// TwinCAT 3 PLC project test
// ProgramVersion: 3.1.4020.5
// libraries:
//   LCLS General, * (SLAC)
//   LCLS Vacuum, * (SLAC - LCLS)
//   PMPS, * (SLAC - LCLS)
//   Tc2_Standard, * (Beckhoff Automation GmbH)
//   Tc2_System, * (Beckhoff Automation GmbH)
//   Tc2_Utilities, * (Beckhoff Automation GmbH)
//   Tc3_Module, * (Beckhoff Automation GmbH)
// project tree:
//   DUTs/ E_STATES.TcTLEO (not stored)
//   functions/ FB_TurboExtLogic.TcPOU, F_RoughPumpInlet_ILK.TcPOU, F_TurboExtILKLogic.TcPOU, F_TurboExtILKLogic_2.TcPOU, F_TurboExtILK_NO.TcPOU, F_TurboExtILK_NO_T.TcPOU, F_TurboGateValve_ILK.TcPOU, F_TurboGateValve_ILK_1.TcPOU (not stored), F_TurboGateValve_Protection_ILK.TcPOU, F_TURBO_VRC_ILK.TcPOU, F_VALVE_REL_ILK.TcPOU (not stored), F_VRC_DIODE_ILK.TcPOU, F_VRC_DIODE_ILK_OK.TcPOU
//   GVLs/ GVL_Devices.TcGVL, GVL_PMPS.TcGVL
//   / PlcTask.TcTTO (not stored)
//   POUs/ FB_VGC_tst.TcPOU, MAIN.TcPOU
// real-time tasks:
//   TASK PlcTask: cycle T#10ms, priority 20, ADS port 350
//   TASK SimTask: cycle T#10ms, priority 1, ADS port 351
//   TASK VacTask: cycle T#10ms, priority 2, ADS port 352
// I/O:
//   DEVICE Device 1 (EtherCAT) (disabled), AmsNetId 172.21.148.60.2.1
//     Term 1 (EK1100) [EK1100 EtherCAT Coupler (2A E-Bus)]
//       Term 2 (EL3174-0002) [EL3174-0002 4Ch. Ana. Input +/-10V, +/-20mA 16 Bit, Isolated Channels]
//       Term 3 (EL3174-0002) [EL3174-0002 4Ch. Ana. Input +/-10V, +/-20mA 16 Bit, Isolated Channels]
//       Term 4 (EL2624) [EL2624 4Ch. Relay Output, NO (125V AC / 30V DC)]
//       Term 6 (EL1004) [EL1004 4Ch. Dig. Input 24V, 3ms]
//       Term 5 (EL1004) [EL1004 4Ch. Dig. Input 24V, 3ms]
//       Term 7 (EL2004) [EL2004 4Ch. Dig. Output 24V, 0.5A]
//       Term 8 (EL3064) [EL3064 4Ch. Ana. Input 0-10V]
//       Term 9 (EL2794) [EL2794 4Ch. Dig. Output 24V AC/DC, 2A, short-circuit-proof]
//       Term 10 (EL1004) [EL1004 4Ch. Dig. Input 24V, 3ms]
//       Term 11 (EL1124) [EL1124 4Ch. Dig. Input 5V, 10µs, Sensor Power]
//       Term 12 (EL1124) [EL1124 4Ch. Dig. Input 5V, 10µs, Sensor Power]
//       Term 13 (EL3064) [EL3064 4Ch. Ana. Input 0-10V]
// variable links:
//   SIM/SIM Instance <-> test/test Instance
//     PlcTaskSim Inputs/GVL_SimDevices.PMPS_VGC_01.i_xSol <-> PlcTask Outputs/GVL_Devices.PMPS_VGC_01.q_xOPN_DO
//     PlcTaskSim Inputs/GVL_SimDevices.PMPS_VGC_02.i_xSol <-> PlcTask Outputs/GVL_Devices.PMPS_VGC_02.q_xOPN_DO
//     PlcTaskSim Inputs/GVL_SimDevices.PMPS_VGC_03.i_xSol <-> PlcTask Outputs/GVL_Devices.PMPS_VGC_03.q_xOPN_DO
//     PlcTaskSim Inputs/GVL_SimDevices.PMPS_VGC_04.i_xSol <-> PlcTask Outputs/GVL_Devices.PMPS_VGC_04.q_xOPN_DO
//     PlcTaskSim Inputs/GVL_SimDevices.PMPS_VGC_05.i_xSol <-> PlcTask Outputs/GVL_Devices.PMPS_VGC_05.q_xOPN_DO
//     PlcTaskSim Inputs/GVL_SimDevices.PMPS_VGC_06.i_xSol <-> PlcTask Outputs/GVL_Devices.PMPS_VGC_06.q_xOPN_DO
//     PlcTaskSim Inputs/GVL_SimDevices.PMPS_VGC_08.i_xSol <-> PlcTask Outputs/GVL_Devices.PMPS_VGC_08.q_xOPN_DO
//     PlcTaskSim Inputs/GVL_SimDevices.PMPS_VGC_09.i_xSol <-> PlcTask Outputs/GVL_Devices.PMPS_VGC_09.q_xOPN_DO
//     PlcTaskSim Inputs/GVL_SimDevices.PMPS_VGC_10.i_xSol <-> PlcTask Outputs/GVL_Devices.PMPS_VGC_10.q_xOPN_DO
//     PlcTaskSim Inputs/GVL_SimDevices.PMPS_VGC_11.i_xSol <-> PlcTask Outputs/GVL_Devices.PMPS_VGC_11.q_xOPN_DO
//     PlcTaskSim Inputs/GVL_SimDevices.S_FEE_GCC_03.i_xHvOn <-> PlcTask Outputs/GVL_Devices.FEE_GCC_03.q_xHV_DIS
//     PlcTaskSim Inputs/GVL_SimDevices.S_FEE_GCC_04.i_xHvOn <-> PlcTask Outputs/GVL_Devices.FEE_GCC_04.q_xHV_DIS
//     PlcTaskSim Inputs/GVL_SimDevices.S_FEE_KMONO_GCC_01.i_xHvOn <-> PlcTask Outputs/GVL_Devices.FEE_KMONO_GCC_01.q_xHV_DIS
//     PlcTaskSim Inputs/GVL_SimDevices.S_FEE_KMONO_PIP_01.xOn <-> PlcTask Outputs/GVL_Devices.FEE_KMONO_PIP_01.q_xHVEna_DO
//     PlcTaskSim Inputs/GVL_SimDevices.S_FEE_M1L_PIP_01.xOn <-> PlcTask Outputs/GVL_Devices.FEE_M1L_PIP_01.q_xHVEna_DO
//     PlcTaskSim Inputs/GVL_SimDevices.S_FEE_MIL_GCC_02.i_xHvOn <-> PlcTask Outputs/GVL_Devices.FEE_M1L_GCC_01.q_xHV_DIS
//     PlcTaskSim Inputs/GVL_SimDevices.S_FEE_PIP_02.xOn <-> PlcTask Outputs/GVL_Devices.FEE_PIP_02.q_xHVEna_DO
//     PlcTaskSim Inputs/GVL_SimDevices.S_FEE_PIP_03.xOn <-> PlcTask Outputs/GVL_Devices.FEE_PIP_03.q_xHVEna_DO
//     PlcTaskSim Inputs/GVL_SimDevices.S_FEE_VGC_02.i_xSol <-> PlcTask Outputs/GVL_Devices.FEE_VGC_02.q_xOPN_DO
//     PlcTaskSim Inputs/GVL_SimDevices.VGC_2S.i_xSol <-> PlcTask Outputs/MAIN.VGC_2S.q_xOPN_DO
//     PlcTaskSim Outputs/GVL_SimDevices.PMPS_VGC_01.q_xClsLS <-> PlcTask Inputs/GVL_Devices.PMPS_VGC_01.i_xClsLS
//     PlcTaskSim Outputs/GVL_SimDevices.PMPS_VGC_02.q_xClsLS <-> PlcTask Inputs/GVL_Devices.PMPS_VGC_02.i_xClsLS
//     PlcTaskSim Outputs/GVL_SimDevices.PMPS_VGC_03.q_xClsLS <-> PlcTask Inputs/GVL_Devices.PMPS_VGC_03.i_xClsLS
//     PlcTaskSim Outputs/GVL_SimDevices.PMPS_VGC_04.q_xClsLS <-> PlcTask Inputs/GVL_Devices.PMPS_VGC_04.i_xClsLS
//     PlcTaskSim Outputs/GVL_SimDevices.PMPS_VGC_05.q_xClsLS <-> PlcTask Inputs/GVL_Devices.PMPS_VGC_05.i_xClsLS
//     PlcTaskSim Outputs/GVL_SimDevices.PMPS_VGC_06.q_xClsLS <-> PlcTask Inputs/GVL_Devices.PMPS_VGC_06.i_xClsLS
//     PlcTaskSim Outputs/GVL_SimDevices.PMPS_VGC_08.q_xClsLS <-> PlcTask Inputs/GVL_Devices.PMPS_VGC_08.i_xClsLS
//     PlcTaskSim Outputs/GVL_SimDevices.PMPS_VGC_09.q_xClsLS <-> PlcTask Inputs/GVL_Devices.PMPS_VGC_09.i_xClsLS
//     PlcTaskSim Outputs/GVL_SimDevices.PMPS_VGC_10.q_xClsLS <-> PlcTask Inputs/GVL_Devices.PMPS_VGC_10.i_xClsLS
//     PlcTaskSim Outputs/GVL_SimDevices.PMPS_VGC_11.q_xClsLS <-> PlcTask Inputs/GVL_Devices.PMPS_VGC_11.i_xClsLS
//     PlcTaskSim Outputs/GVL_SimDevices.PMPS_VGC_01.q_xOpnLS <-> PlcTask Inputs/GVL_Devices.PMPS_VGC_01.i_xOpnLS
//     PlcTaskSim Outputs/GVL_SimDevices.PMPS_VGC_02.q_xOpnLS <-> PlcTask Inputs/GVL_Devices.PMPS_VGC_02.i_xOpnLS
//     PlcTaskSim Outputs/GVL_SimDevices.PMPS_VGC_03.q_xOpnLS <-> PlcTask Inputs/GVL_Devices.PMPS_VGC_03.i_xOpnLS
//     PlcTaskSim Outputs/GVL_SimDevices.PMPS_VGC_04.q_xOpnLS <-> PlcTask Inputs/GVL_Devices.PMPS_VGC_04.i_xOpnLS
//     PlcTaskSim Outputs/GVL_SimDevices.PMPS_VGC_05.q_xOpnLS <-> PlcTask Inputs/GVL_Devices.PMPS_VGC_05.i_xOpnLS
//     PlcTaskSim Outputs/GVL_SimDevices.PMPS_VGC_06.q_xOpnLS <-> PlcTask Inputs/GVL_Devices.PMPS_VGC_06.i_xOpnLS
//     PlcTaskSim Outputs/GVL_SimDevices.PMPS_VGC_08.q_xOpnLS <-> PlcTask Inputs/GVL_Devices.PMPS_VGC_08.i_xOpnLS
//     PlcTaskSim Outputs/GVL_SimDevices.PMPS_VGC_09.q_xOpnLS <-> PlcTask Inputs/GVL_Devices.PMPS_VGC_09.i_xOpnLS
//     PlcTaskSim Outputs/GVL_SimDevices.PMPS_VGC_10.q_xOpnLS <-> PlcTask Inputs/GVL_Devices.PMPS_VGC_10.i_xOpnLS
//     PlcTaskSim Outputs/GVL_SimDevices.PMPS_VGC_11.q_xOpnLS <-> PlcTask Inputs/GVL_Devices.PMPS_VGC_11.i_xOpnLS
//     PlcTaskSim Outputs/GVL_SimDevices.S_FEE_GCC_03.q_DisActive <-> PlcTask Inputs/GVL_Devices.FEE_GCC_03.i_xDisc_Active
//     PlcTaskSim Outputs/GVL_SimDevices.S_FEE_GCC_04.q_DisActive <-> PlcTask Inputs/GVL_Devices.FEE_GCC_04.i_xDisc_Active
//     PlcTaskSim Outputs/GVL_SimDevices.S_FEE_GCC_03.q_iRawPress <-> PlcTask Inputs/GVL_Devices.FEE_GCC_03.i_iPRESS_R
//     PlcTaskSim Outputs/GVL_SimDevices.S_FEE_GCC_04.q_iRawPress <-> PlcTask Inputs/GVL_Devices.FEE_GCC_04.i_iPRESS_R
//     PlcTaskSim Outputs/GVL_SimDevices.S_FEE_GCC_03.q_xHVOn <-> PlcTask Inputs/GVL_Devices.FEE_GCC_03.i_xHV_ON
//     PlcTaskSim Outputs/GVL_SimDevices.S_FEE_GCC_04.q_xHVOn <-> PlcTask Inputs/GVL_Devices.FEE_GCC_04.i_xHV_ON
//     PlcTaskSim Outputs/GVL_SimDevices.S_FEE_GPI_03.q_iRawPress <-> PlcTask Inputs/GVL_Devices.FEE_GPI_03.i_iPRESS_R
//     PlcTaskSim Outputs/GVL_SimDevices.S_FEE_GPI_04.q_iRawPress <-> PlcTask Inputs/GVL_Devices.FEE_GPI_04.i_iPRESS_R
//     PlcTaskSim Outputs/GVL_SimDevices.S_FEE_KMONO_GCC_01.q_DisActive <-> PlcTask Inputs/GVL_Devices.FEE_KMONO_GCC_01.i_xDisc_Active
//     PlcTaskSim Outputs/GVL_SimDevices.S_FEE_KMONO_GCC_01.q_iRawPress <-> PlcTask Inputs/GVL_Devices.FEE_KMONO_GCC_01.i_iPRESS_R
//     PlcTaskSim Outputs/GVL_SimDevices.S_FEE_KMONO_GCC_01.q_xHVOn <-> PlcTask Inputs/GVL_Devices.FEE_KMONO_GCC_01.i_xHV_ON
//     PlcTaskSim Outputs/GVL_SimDevices.S_FEE_KMONO_GPI_01.q_iRawPress <-> PlcTask Inputs/GVL_Devices.FEE_KMONO_GPI_01.i_iPRESS_R
//     PlcTaskSim Outputs/GVL_SimDevices.S_FEE_M1L_GPI_02.q_iRawPress <-> PlcTask Inputs/GVL_Devices.FEE_M1L_GPI_01.i_iPRESS_R
//     PlcTaskSim Outputs/GVL_SimDevices.S_FEE_MIL_GCC_02.q_DisActive <-> PlcTask Inputs/GVL_Devices.FEE_M1L_GCC_01.i_xDisc_Active
//     PlcTaskSim Outputs/GVL_SimDevices.S_FEE_MIL_GCC_02.q_iRawPress <-> PlcTask Inputs/GVL_Devices.FEE_M1L_GCC_01.i_iPRESS_R
//     PlcTaskSim Outputs/GVL_SimDevices.S_FEE_MIL_GCC_02.q_xHVOn <-> PlcTask Inputs/GVL_Devices.FEE_M1L_GCC_01.i_xHV_ON
//     PlcTaskSim Outputs/GVL_SimDevices.S_FEE_VGC_02.q_xClsLS <-> PlcTask Inputs/GVL_Devices.FEE_VGC_02.i_xClsLS
//     PlcTaskSim Outputs/GVL_SimDevices.S_FEE_VGC_02.q_xOpnLS <-> PlcTask Inputs/GVL_Devices.FEE_VGC_02.i_xOpnLS
//     PlcTaskSim Outputs/GVL_SimDevices.VGC_2S.q_xClsLS <-> PlcTask Inputs/MAIN.VGC_2S.i_xClsLS
//     PlcTaskSim Outputs/GVL_SimDevices.VGC_2S.q_xOpnLS <-> PlcTask Inputs/MAIN.VGC_2S.i_xOpnLS

// ---- GVLs/GVL_Devices.TcGVL
VAR_GLOBAL
	
	

/////////////////////
	{attribute 'pytmc' := '
    pv: FEE:VGC:02
	'}
	FEE_VGC_02: FB_VGC;
	{attribute 'pytmc' := '
    pv: FEE:KMONO:GPI:01
	'}
	FEE_KMONO_GPI_01: FB_MKS275;
	{attribute 'pytmc' := '
    pv: FEE:KMONO:GCC:01
	'}
	FEE_KMONO_GCC_01: FB_MKS500;
	{attribute 'pytmc' := '
    pv: FEE:KMONO:PIP:01
	'}
	FEE_KMONO_PIP_01: FB_PIP_Gamma;
	{attribute 'pytmc' := '
    pv: FEE:PIP:02
	'}
	FEE_PIP_02: FB_PIP_Gamma;
	{attribute 'pytmc' := '
    pv: FEE:GPI:03
	'}
	FEE_GPI_03: FB_MKS275;
	{attribute 'pytmc' := '
    pv: FEE:GCC:03
	'}
	FEE_GCC_03: FB_MKS500;
	{attribute 'pytmc' := '
    pv: FEE:VGC:03
	'}
	//FEE_VGC_03: FB_VGC_FFO;
	{attribute 'pytmc' := '
    pv: FEE:M1L:GPI:01
	'}
	FEE_M1L_GPI_01: FB_MKS275;
	{attribute 'pytmc' := '
    pv: FEE:M1L:GCC:03
	'}
	FEE_M1L_GCC_01: FB_MKS500;
	{attribute 'pytmc' := '
    pv: FEE:M1L:PIP:01
	'}
	FEE_M1L_PIP_01: FB_PIP_Gamma;
	{attribute 'pytmc' := '
    pv: FEE:PIP:03
	'}
	FEE_PIP_03: FB_PIP_Gamma;
	{attribute 'pytmc' := '
    pv: FEE:GPI:04
	'}
	FEE_GPI_04: FB_MKS275;
	{attribute 'pytmc' := '
    pv: FEE:GCC:04
	'}
	FEE_GCC_04: FB_MKS500;
	{attribute 'pytmc' := '
    pv: FEE:VGC:04
	'}
	//FEE_VGC_04: FB_VGC_FFO;
	
	PMPS_VGC_01: FB_VGC;
	PMPS_VGC_02: FB_VGC;
	PMPS_VGC_03: FB_VGC;
	PMPS_VGC_04: FB_VGC;
	PMPS_VGC_05: FB_VGC;
	PMPS_VGC_06: FB_VGC;
	
	PMPS_VGC_08: FB_VGC;
	PMPS_VGC_09: FB_VGC;
	
	PMPS_VGC_10: FB_VGC;
	PMPS_VGC_11: FB_VGC;
	
	PTM_Agilent: FB_PTM_Agilent; 
			
	
END_VAR

// ---- GVLs/GVL_PMPS.TcGVL

VAR_GLOBAL
	 g_FastFaultOutput3  :   FB_HardwareFFOutput;
	
{attribute 'pytmc' := '
    pv: PLC:TST:FF1
    '}
    {attribute 'TcLinkTo' := '.q_xFastFaultOut:=TIIB[PMPS_FFO]^Channel 1^Output'}
    g_FastFaultOutput1  :   FB_HardwareFFOutput;
	
	{attribute 'pytmc' := '
    pv: PLC:TST:FF2
    '}
    {attribute 'TcLinkTo' := '.q_xFastFaultOut:=TIIB[PMPS_FFO]^Channel 2^Output'}
    g_FastFaultOutput2  :   FB_HardwareFFOutput;
	
END_VAR

// ---- functions/FB_TurboExtLogic.TcPOU
(*deprecated*)
FUNCTION_BLOCK FB_TurboExtLogic
VAR_IN_OUT
	Turbo		:	ST_AgilentPTM;
END_VAR
VAR_INPUT
	BackingGauge:	ST_VG;
	InletGauge	:	ST_VG;
	VentValve	:	ST_VCC_NO;
	ScrollPump	:	ST_RoughPump;
END_VAR
VAR_OUTPUT
END_VAR
VAR
END_VAR

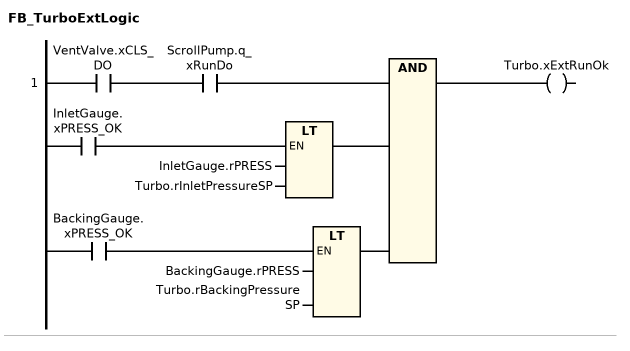
// NETWORK 1
Turbo.xExtRunOk := (VentValve.xCLS_DO AND ScrollPump.q_xRunDo) AND (InletGauge.xPRESS_OK AND InletGauge.rPRESS < Turbo.rInletPressureSP) AND (BackingGauge.xPRESS_OK AND BackingGauge.rPRESS < Turbo.rBackingPressureSP);

END_FUNCTION_BLOCK

// ---- functions/F_RoughPumpInlet_ILK.TcPOU
(*
	Determine whether a pump attached to the inlet of a roughing pump is safe to open. 
	
	Return true, signaling it is safe to open when the roughing pump is confirmed to be working. 
*)

FUNCTION F_RoughPumpInlet_ILK : BOOL
VAR_INPUT
	ScrollPump	:	ST_RoughPump;
END_VAR
VAR
END_VAR


F_RoughPumpInlet_ILK := (ScrollPump.eState = pumpRUNNING); (* Confirm that the roughing pump is running before opening the valve *)

END_FUNCTION

// ---- functions/F_TurboExtILKLogic.TcPOU

(* This function evaluates the Turbo ILK logic*)
(* The Turbo shall not Run if the vent valve is open*)
(* The function also switches off the Turbo if the Inlet pressure or the backing Pressure*)
(* are higher than the configured set point*)
FUNCTION F_TurboExtILKLogic : BOOL
VAR_INPUT
	Turbo		:	ST_PTM;
	BackingGauge:	ST_VG;
	InletGauge	:	ST_VG;
	VentValve	:	ST_VVC;
	ScrollPump	:	ST_RoughPump;
END_VAR

VAR
END_VAR

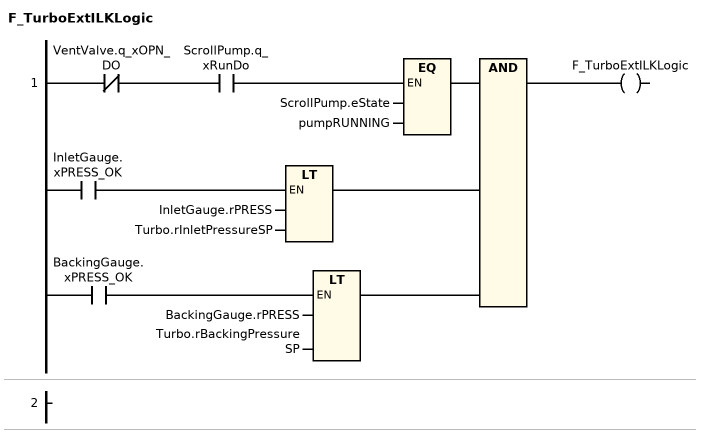
// NETWORK 1
F_TurboExtILKLogic := (NOT VentValve.q_xOPN_DO AND ScrollPump.q_xRunDo AND ScrollPump.eState = pumpRUNNING) AND (InletGauge.xPRESS_OK AND InletGauge.rPRESS < Turbo.rInletPressureSP) AND (BackingGauge.xPRESS_OK AND BackingGauge.rPRESS < Turbo.rBackingPressureSP);

// NETWORK 2

END_FUNCTION

// ---- functions/F_TurboExtILKLogic_2.TcPOU

(* This function evaluates the Turbo ILK logic*)
(* The function switches off the Turbo if the Inlet pressure or the backing Pressure*)
(* are higher than the configured set point*)
FUNCTION F_TurboExtILKLogic_2 : BOOL
VAR_INPUT
	Turbo		:	ST_PTM;
	BackingGauge:	ST_VG;
	InletGauge	:	ST_VG;
	ScrollPump	:	ST_RoughPump;
END_VAR
VAR
END_VAR

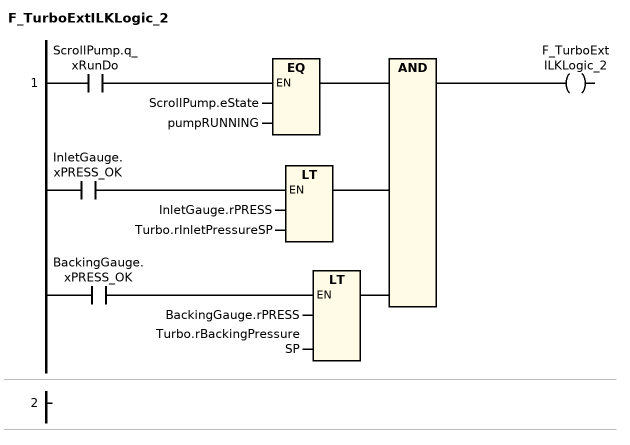
// NETWORK 1
F_TurboExtILKLogic_2 := (ScrollPump.q_xRunDo AND ScrollPump.eState = pumpRUNNING) AND (InletGauge.xPRESS_OK AND InletGauge.rPRESS < Turbo.rInletPressureSP) AND (BackingGauge.xPRESS_OK AND BackingGauge.rPRESS < Turbo.rBackingPressureSP);

// NETWORK 2

END_FUNCTION

// ---- functions/F_TurboExtILK_NO.TcPOU
(* This function Block interfaces with a NO turbo valve*)
(* Mainly used in the FEE HXR GATT*)
FUNCTION F_TurboExtILK_NO : BOOL
VAR_INPUT
	Turbo		:	ST_PTM;
	BackingGauge:	ST_VG;
	InletGauge	:	ST_VG;
	VentValve	:	ST_VCC_NO; //NO type turbo valve
	ScrollPump	:	ST_RoughPump;
	Timer :TON;
END_VAR

VAR
END_VAR
VAR // added by the converter: edge detectors and wires of the graphical bodies
    _w1 : BOOL;
END_VAR

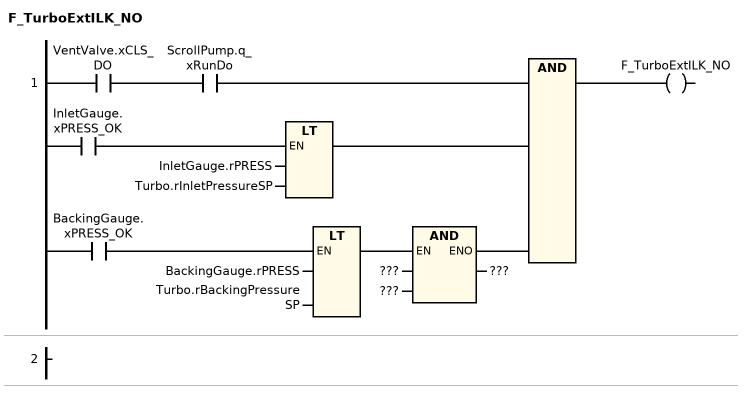
// NETWORK 1
_w1 := BackingGauge.xPRESS_OK AND BackingGauge.rPRESS < Turbo.rBackingPressureSP;
IF _w1 THEN (* ??? AND ???; result not used *) END_IF
F_TurboExtILK_NO := (VentValve.xCLS_DO AND ScrollPump.q_xRunDo) AND (InletGauge.xPRESS_OK AND InletGauge.rPRESS < Turbo.rInletPressureSP) AND _w1;

// NETWORK 2

END_FUNCTION

// ---- functions/F_TurboExtILK_NO_T.TcPOU
FUNCTION F_TurboExtILK_NO_T : BOOL
VAR_INPUT
	Turbo		:	ST_PTM;
	BackingGauge:	ST_VG;
	InletGauge	:	ST_VG;
	VentValve	:	ST_VCC_NO; //NO type turbo valve
	ScrollPump	:	ST_RoughPump;
END_VAR
VAR
	Timer :TON;
END_VAR

END_FUNCTION

// ---- functions/F_TurboGateValve_ILK.TcPOU
(* This Function Block evaluates the ILK condition of the Turbo Gate valve *)
(* The logic Protects the Turbo pump from inlet pressure above the SP*)

FUNCTION F_TurboGateValve_ILK : BOOL (* function return TRUE when ILK is OK*)
VAR_INPUT
	i_Turbo : ST_PTM; // Turbo Pump
	i_stISG : ST_VG; //Gauge measuring inlet Pressure e.g Pirani
END_VAR
VAR
END_VAR

(* This Function Block evaluates the ILK condition of the Turbo Gate valve *)
(* The logic Protects the Turbo pump from inlet pressure above the SP*)
F_TurboGateValve_ILK := (NOT (i_Turbo.eState = pumpSTOPPED) AND NOT (i_Turbo.eState = pumpSTOPPING) AND NOT (i_Turbo.eState = pumpFAULT))
						AND (i_stISG.xPRESS_OK AND i_stISG.rPRESS < i_Turbo.rInletPressureSP);

END_FUNCTION

// ---- functions/F_TurboGateValve_Protection_ILK.TcPOU
(* This Function Block evaluates the ILK condition of the Turbo Gate valve *)
(* The logic Protects the Turbo pump from inlet pressure above the SP*)
(* And Protects the Turbo pump from backing pressure above the SP*)
(* And Protects the Turbo pump in the case of backing pump not running*)

FUNCTION F_TurboGateValve_Protection_ILK : BOOL (* function return TRUE when ILK is OK*)
VAR_INPUT
	i_Turbo : ST_PTM; // Turbo Pump
	i_stISG : ST_VG; //Gauge measuring inlet Pressure e.g Pirani
	i_stBSG : ST_VG; //Gauge measuring backing Pressure e.g Pirani
	ScrollPump	:	ST_RoughPump; // Roughing pump
END_VAR
VAR
END_VAR

(* This Function Block evaluates the ILK condition of the Turbo Gate valve *)
(* The logic Protects the Turbo pump from inlet pressure above the SP*)
F_TurboGateValve_Protection_ILK := (NOT (i_Turbo.eState = pumpSTOPPED) AND NOT (i_Turbo.eState = pumpSTOPPING) AND NOT (i_Turbo.eState = pumpFAULT))
						AND (i_stISG.xPRESS_OK AND i_stISG.rPRESS < i_Turbo.rInletPressureSP)
						AND (i_stBSG.xPRESS_OK AND i_stBSG.rPRESS < i_Turbo.rBackingPressureSP)
						AND (ScrollPump.eState = pumpRUNNING);

END_FUNCTION

// ---- functions/F_TURBO_VRC_ILK.TcPOU
(* Close the vic if the roughing pump pirani loses its at-vac setpoint while the turbo is pumping *)
FUNCTION F_TURBO_VRC_ILK : BOOL
VAR_INPUT

	i_xHiVac 	: BOOL;
	i_xRunPTM	: BOOL;
	i_xFLVac	: BOOL;

END_VAR
VAR

	rHysterisis : REAL := 0;

	xInterlock: BOOL;
	rTolerance: REAL := 20;
END_VAR

(* Close the vic if the roughing pump pirani loses its at-vac setpoint while the turbo is pumping *)
F_TURBO_VRC_ILK := (NOT i_xHiVac AND NOT i_xRunPTM AND NOT i_xFLVac) OR
					(NOT i_xRunPTM AND i_xFLVac) OR
					(i_xRunPTM AND i_xFLVac);

END_FUNCTION

// ---- functions/F_VRC_DIODE_ILK.TcPOU
(* The principle is simple, a VRC should never open when B side pressure is greater than 
the A side pressure. *)

FUNCTION F_VRC_DIODE_ILK : BOOL
VAR_INPUT

	i_stPGA : ST_VG; // A side pressure gauge
	i_stPGB	: ST_VG; // B side pressure gauge

END_VAR
VAR

	rHysterisis : REAL := 0;

	xInterlock: BOOL;
	rTolerance: REAL := 20;
END_VAR

(* The principle is simple, a VRC should never open when B side pressure is greater than the A side pressure. *)
rTolerance := 20;
F_VRC_DIODE_ILK := ((i_stPGA.rPRESS + rTolerance >= i_stPGB.rPRESS + rHysterisis) OR i_stPGA.xBAKEOUT) AND i_stPGA.xPRESS_OK AND i_stPGB.xPRESS_OK;

(* OK it gets a bit more complicated with hysterisis,

Now, if the F_VIC_DIODE_ILK is FALSE then some hysterisis is added to the B side. But if it's OK then we just stick with making sure that the A side is greater than the B side

*)
(*
IF NOT F_VIC_DIODE_ILK THEN
Hysterisis := 40;
ELSE
Hysterisis := 0;
END_IF
*)

END_FUNCTION

// ---- functions/F_VRC_DIODE_ILK_OK.TcPOU
(*The function returns TRUE i.e. ILK_OK when pressure on A side is greater than or equal to the pressure on B side*)
FUNCTION F_VRC_DIODE_ILK_OK : BOOL
VAR_INPUT

	i_stPGA : ST_VG; // A side pressure gauge
	i_stPGB	: ST_VG; // B side pressure gauge

END_VAR
VAR
	rHysterisis : REAL := 0;

	xInterlock: BOOL;
	rTolerance: REAL := 0;
END_VAR

(* The principle is simple, a VRC should never open when B side pressure is greater than the A side pressure. *)
F_VRC_DIODE_ILK_OK := (i_stPGA.rPRESS + rTolerance >= i_stPGB.rPRESS + rHysterisis) AND i_stPGA.xPRESS_OK AND i_stPGB.xPRESS_OK;

END_FUNCTION

// ---- POUs/FB_VGC_tst.TcPOU
(* This function block implements basic functionality for Isolation Gate Valves*)
(* This function block interlock is as follows:
1. The valve can be opened when the difference between the pressures on both sides is
less than the maximum differential pressure.
2. This rule persists until the pressures on both sides are lower than the vacuum-setpoint.
3. Once at-vac, the valve will close if the pressure on either side rises above the setpoint.*)
(*This function block also implements PMPS and EPS interlocks, as well as Fast MPS trigger*)
{attribute 'no_check'}
{attribute 'reflection'} 
FUNCTION_BLOCK FB_VGC_tst Extends FB_Valve
VAR_IN_OUT
	
END_VAR
VAR_INPUT
	(*Upstream Gauge, usually ion gauge*)
	i_stUSG	:	ST_VG;
	(*Downstream Gauge, usually ion gauge*)
	i_stDSG	:	ST_VG;
	{attribute 'pytmc' := '
    pv: Dis_DPIlk
	'}
	i_xDis_DPIlk : BOOL := FALSE;  (* Set to true when calling the function to disable the differential pressure interlock *)
	i_xPMPS_OK:	BOOL	; (*Set to True To switch of the bptm*)
	{attribute 'pytmc' := '
    pv: EPS_OK
	'}
	i_xEPS_OK:	BOOL	:= TRUE; (*External EPS interlock, Set to TRUE when no EPS interlock is required, otherwise set to correct interlock signal*)
	i_xExt_OK: BOOL; (*Other External Interlock, Set to True when no external interlock is required. If this Valve is neigboring a Fast Shutter this should be linked to the fast shutter xVAC_FAULT_OK*)
	i_xOverrideMode : BOOL; (*To be linked to global override bit. This Overrides Vacuum logic only, EPS, MPS and PMPS are still enforces*)
	// Reset fault
	{attribute 'pytmc' := '
    pv: FF_Reset
	'}
    i_xReset: BOOL;
	i_xIsAperture:BOOL :=FALSE; // Set tp True if this is an Aperture Valve, the MPS Fault will trip only when moving.
	i_sDevName : T_MaxString :=  'VGC'; // Device name for diagnostic
	i_nTransitionRootID: UDINT; //A unique transition Root ID that is equal to or greater than 1000
END_VAR
VAR_OUTPUT
	{attribute 'pytmc' := '
    pv:
	'}
	iq_stValve : ST_VGC; (* All valve data and states will be in this struct*)
	
	{attribute 'pytmc' := '
    pv: MPS_FAULT_OK
	field: ZNAM MPS FAULT ;
	field: ONAM MPS OK ;
	'}
	xMPS_OK:	BOOL; (*MPS Fast OK, is set when the Valve is Open*)
END_VAR
VAR_IN_OUT
	io_fbFFHWO    :    FB_HardwareFFOutput;
	fbArbiter: FB_Arbiter();
END_VAR
VAR
	// PMPS
	{attribute 'pytmc' := '
    pv: MPS_OK
	'}
	xPMPS_OK:	BOOL	; (*PMPS interlock*)
	bMoving : BOOL;
	bDone :BOOL;
	tBPTMtimeout:TON;
	 i_nRequestedAssertionID:DWORD;
	bptm: BeamParameterTransitionManager;  
	FFO    :    FB_FastFault :=(
        i_DevName := 'VGC',
        i_Desc := 'Fault occurs when the valve is not in open state',
        i_TypeCode := 16#1010);
	//g_FastFaultOutput1	:	FB_HardwareFFOutput;	

	{attribute 'instance-path'}
	{attribute 'noinit'}
	sPath: STRING;
	
	rDiffPressAllowed	:	REAL := 22.5; // Torr, Default value comes from Vat Valve Manual
	rDiffPress : REAL;
	set : BOOL;
    reset: BOOL;
	  
	xFirstPass	:	BOOL;
	fbFSInit		:	R_TRIG;
	
	tonDelOK : TON;
	rtOK	:	R_TRIG;
	tonOvrd	:	TON;
	rtOpen	:	R_TRIG;
	ftClose: F_TRIG;
	
	tDelOK	:	TIME := T#60S;
	tOvrd	:	TIME := T#10s;
	
	
	(* Timeouts*)
	tTimeOutDuration: TIME:= T#30S;
	tOPNtimeout: TON;
	tCLStimeout:TON;
	
	
	(*IO*)
	i_xOpnLS	AT%I*: BOOL;
	i_xClsLS	AT%I*: BOOL;
	q_xOPN_DO	AT%Q*: BOOL;
    
    // For logging
    eVGCPrevState : E_VGC;
 
	
END_VAR

(* Vacuum gate valve
A. Wallace
16-10-29

A gate valve isolates vacuum volumes. Ideally it can be opened when a system is vented
to allow for faster pumping, and will close when high vacuum is lost.

The following behavior is good for valves in something like a gas attenuator.
This function block does the following:
1. The valve can be opened when the difference between the pressures on both sides is
less than the maximum differential pressure.
2. This rule persists until the pressures on both sides are lower than the vacuum-setpoint.
3. Once at-vac, the valve will close if the pressure on either side rises above the setpoint.

Alternatively, the differential pressure interlock can be disabled so the valve may only be opened
if the pressure on both sides is lower than the at-vacuum-setpoint. You want this behavior if 
the valve is to be used in a UHV section.

Hysteresis is employed to ensure a smooth transition from vented/pumping down, to at-vac.

Finally, an override system is built in so you can bypass all the interlocking logic and 
get back online.
*)
(* 10/1/2018 Margaret Ghaly included EPS, PMPS Checkes and MPS trigger signals*)


fbFSInit( CLK := TRUE, Q => xFirstPass);
(*IO Mapping*)
ACT_IO();

(* On first PLC pass, put valve into vented state, which implies a closed valve *)
IF xFirstPass THEN
	iq_stValve.eVGC_State := Vented;
	iq_stValve.pv_xOPN_SW := FALSE;
	FFO.i_DevName := i_sDevName;
END_IF


///Check valve position
IF iq_stValve.i_xClsLS AND  iq_stValve.i_xOpnLS THEN
	iq_stValve.eState:=INVALID;
ELSIF NOT iq_stValve.i_xClsLS AND iq_stValve.i_xOpnLS AND iq_stValve.q_xOPN_DO THEN 
	iq_stValve.eState:=OPEN;
ELSIF NOT iq_stValve.i_xClsLS AND iq_stValve.i_xOpnLS AND NOT iq_stValve.q_xOPN_DO THEN 
	iq_stValve.eState:=OPEN_F;
ELSIF iq_stValve.i_xClsLS AND NOT iq_stValve.i_xOpnLS AND NOT iq_stValve.q_xOPN_DO THEN 
	iq_stValve.eState:=CLOSED;
ELSIF NOT iq_stValve.i_xClsLS AND NOT iq_stValve.i_xOpnLS THEN 
	iq_stValve.eState:=MOVING;
ELSE
	iq_stValve.eState:=INVALID;
END_IF

// Update hysteresis
///////////////////////////////////////////////////
IF iq_stValve.rAT_VAC_SP_LAST <> iq_stValve.rAT_VAC_SP OR xFirstPass THEN
	iq_stValve.rAT_VAC_SP_LAST := iq_stValve.rAT_VAC_SP;
	iq_stValve.rAT_VAC_HYS := iq_stValve.rHYST_PERC * iq_stValve.rAT_VAC_SP;
END_IF

iq_stValve.rAT_VAC_HYS := LIMIT(0, iq_stValve.rAT_VAC_HYS, iq_stValve.rAT_VAC_SP);
IF iq_stValve.rAT_VAC_SP <> 0 THEN
	IF iq_stValve.rHYST_PERC <> (iq_stValve.rAT_VAC_HYS / iq_stValve.rAT_VAC_SP) THEN
		iq_stValve.rHYST_PERC := LIMIT(0, (iq_stValve.rAT_VAC_HYS / iq_stValve.rAT_VAC_SP) ,1);
	END_IF
END_IF
// Valve at vacuum check
///////////////////////////////////////////////////
	set := i_stUSG.rPRESS < iq_stValve.rAT_VAC_HYS AND i_stDSG.rPRESS < iq_stValve.rAT_VAC_HYS AND i_stUSG.xPRESS_OK AND i_stDSG.xPRESS_OK;
 	iq_stValve.xAT_VAC S= set;
	reset := i_stUSG.rPRESS > iq_stValve.rAT_VAC_SP OR i_stDSG.rPRESS > iq_stValve.rAT_VAC_SP OR NOT i_stUSG.xPRESS_OK OR NOT i_stDSG.xPRESS_OK;
	iq_stValve.xAT_VAC R= reset;
	
// Differential pressure check
///////////////////////////////////////////////////
	(* Calc the differential pressure across the valve *)
	rDiffPress := ABS(i_stUSG.rPRESS - i_stDSG.rPRESS);
	
	(* As long as the differential pressure is less than 30mbar, the valve is allowed to open *)
	IF rDiffPress <= rDiffPressAllowed AND i_stUSG.xPRESS_OK AND i_stDSG.xPRESS_OK THEN
		iq_stValve.xDP_OK := TRUE;
	ELSE
		iq_stValve.xDP_OK	:= FALSE;
		(* If the differential pressure is exceeded, even when the valve is open,
		the state is unexpected and triggers a fault, because it suggests that something
		is wrong with the valve, or gauges or mapping or there is a major leak on one side.*)
		iq_stValve.eVGC_State := ERR_DiffPress;
        iq_stValve.xERR_DifPres := TRUE;
	END_IF

// Valve state
///////////////////////////////////////////////////
CASE iq_stValve.eVGC_State OF
	Vented: (* The Vented state is used during pump down *)        
		(* Assuming the pump down went well, we are now at vacuum on both sides,
		so we move to the vacuum state, otherwise remain in the vented state *)
		IF iq_stValve.xAT_VAC AND (NOT (iq_stValve.xERR_DifPres)) AND (NOT (iq_stValve.xERR_SP)) AND (NOT (iq_stValve.xERR_ExtFault))THEN
		    iq_stValve.eVGC_State := AtVacuum;
		ELSE
		    iq_stValve.eVGC_State := Vented;
		END_IF
	
	AtVacuum:
		IF iq_stValve.xAT_VAC THEN
		(* If both pressure setpoints are made,
		then enable the differential pressure interlock, regardless of the valve state
		assuming we're using some kind of ion gauge where a pressure setpoint cannot be higher than 1E-4 T *)
		iq_stValve.eVGC_State := AtVacuum;
				
		ELSE
		
			(* If the valve is open (or in an unknown state) and either gauge is not at it's vacuum setpoint,
			we have a loss of vacuum error *)
			IF (iq_stValve.i_xOpnLS OR (NOT iq_stValve.i_xOpnLS AND NOT iq_stValve.i_xClsLS)) THEN
				iq_stValve.eVGC_State := ERR_LostVac;
				iq_stValve.xERR_SP := TRUE; //TAW changed this to the ERR_SP bool because I think that's what it was intended to be?
		
			(* Alternatively, if the valve is already closed and we lose pressure on one side,
			it was probably intentional venting, so we calmly move back to venting mode, and
			disable the differential pressure interlock *) //?? 
			ELSIF iq_stValve.i_xClsLS THEN
				iq_stValve.eVGC_State := Vented;
			END_IF
		
		END_IF
	
	ERR_DiffPress:       
		IF NOT (iq_stValve.xERR_DifPres) THEN
			IF iq_stValve.xAT_VAC AND (NOT (iq_stValve.xERR_DifPres)) AND (NOT (iq_stValve.xERR_SP)) AND (NOT (iq_stValve.xERR_ExtFault))THEN
		    	iq_stValve.eVGC_State := AtVacuum;
			ELSE
		    	iq_stValve.eVGC_State := Vented;
			END_IF
		END_IF
		
	
	ERR_LostVac:
		IF NOT (iq_stValve.xERR_SP) THEN
			IF iq_stValve.xAT_VAC AND (NOT (iq_stValve.xERR_DifPres)) AND (NOT (iq_stValve.xERR_SP)) AND (NOT (iq_stValve.xERR_ExtFault))THEN
		    	iq_stValve.eVGC_State := AtVacuum;
			ELSE
		    	iq_stValve.eVGC_State := Vented;
			END_IF
		END_IF
		
	ERR_ExtFault:
		IF NOT (iq_stValve.xERR_ExtFault) AND (i_xExt_OK) THEN
			IF iq_stValve.xAT_VAC AND (NOT (iq_stValve.xERR_DifPres)) AND (NOT (iq_stValve.xERR_SP)) AND (NOT (iq_stValve.xERR_ExtFault))THEN
		    	iq_stValve.eVGC_State := AtVacuum;
			ELSE
		    	iq_stValve.eVGC_State := Vented;
			END_IF
		END_IF
END_CASE

IF (NOT i_xExt_OK) AND (iq_stValve.eState=OPEN)  THEN
	iq_stValve.eVGC_State := ERR_ExtFault;
	iq_stValve.xERR_ExtFault := TRUE;
END_IF

// Interlock evaluation - with bypass for DP ILK bypass
///////////////////////////////////////////////
IF i_xDis_DPIlk THEN
	iq_stValve.xOPN_OK := iq_stValve.xEXT_OK; // AND iq_stValve.xDP_OK ;
ELSE
	iq_stValve.xOPN_OK := iq_stValve.xEXT_OK AND iq_stValve.xAT_VAC;
END_IF


(* Valve operation *)

(* Override logic *)
(* Goal: give ability to override, but do so in a way that people won't forget it.
Solution: Override only after ten seconds of override, protect against blips,
when the valve permission goes true for more than ten seconds consistently, remove override
*)

tonDelOK(IN:=iq_stValve.xOPN_OK, PT:=tDelOK);
rtOK(CLK:=tonDelOK.Q);
IF rtOK.Q AND iq_stValve.pv_xOvrdOpn THEN 
	iq_stValve.pv_xOvrdOpn :=FALSE;
	if (iq_stValve.eState = OPEN) AND (i_xOverrideMode) THEN iq_stValve.pv_xOPN_SW := TRUE; END_IF //for seamless transition   
    //Log
    fbLogger(sMsg:='Override expired', eSevr:=TcEventSeverity.Warning);
END_IF
// Release the Force Open bit when the system override is false
IF NOT (i_xOverrideMode) THEN  iq_stValve.pv_xOvrdOpn :=FALSE; END_IF
//Override timer
tonOvrd(IN:=iq_stValve.pv_xOvrdOpn, PT:=tOvrd);


(* Valve operation *)
(* Here's where we evaluate sw actions and operate the valve *)
(* Valve operation *)

ftClose(CLK:= iq_stValve.pv_xOPN_SW);
rtOpen(CLK:= iq_stValve.pv_xOPN_SW);

(*PMPS OPERATION AND BPTM*)
(*PMPS*)
IF NOT(i_xPMPS_OK) THEN
	ACT_PMPS();
END_IF
xPMPS_OK := i_xPMPS_OK OR (bptm.q_xTransitionAuthorized OR tBPTMtimeout.Q);
(*when interlock is lost the Valve closes regardless of the status of the PMPS and EPS*)
IF NOT (iq_stValve.xOPN_OK) THEN
	iq_stValve.pv_xOPN_SW:= FALSE; // Reset switch after inlk is lost
	iq_stValve.q_xOPN_DO := (iq_stValve.pv_xOPN_SW  AND iq_stValve.xOPN_OK) OR (tonOvrd.Q AND i_xOverrideMode);
ELSIF xPMPS_OK THEN 
	iq_stValve.q_xOPN_DO := (iq_stValve.pv_xOPN_SW  AND iq_stValve.xOPN_OK) OR (tonOvrd.Q AND i_xOverrideMode);
END_IF

(*MPS Fault setting*)
If (i_xIsAperture ) THEN 
	(* When the valve  is open or in Closed position MPS is OK, Fault while moving*)
	xMPS_OK := i_xOpnLS XOR i_xClsLS; 
ELSE
	(* When the valve  is open MPS is OK*)
	xMPS_OK := i_xOpnLS AND NOT i_xClsLS AND q_xOPN_DO; 
END_IF


///Check valve moving postion timout
IF NOT iq_stValve.i_xClsLS AND tCLStimeout.Q THEN 
	iq_stValve.bErrorPresent := TRUE;
	iq_stValve.sErrorMessage := 'Close Timeout';
ELSIF NOT iq_stValve.i_xOpnLS AND tOPNtimeout.Q THEN 
	iq_stValve.bErrorPresent := TRUE; 
	iq_stValve.sErrorMessage := 'Open Timeout';
END_IF
IF (iq_stValve.eState=INVALID) THEN
	iq_stValve.bErrorPresent := TRUE; 
	iq_stValve.sErrorMessage := CONCAT(sPath,'Invalid Valve Position');
END_IF


(*Timers*)
tOPNtimeout(IN:= iq_stValve.q_xOPN_DO, PT := tTimeOutDuration );
tCLStimeout(IN:= NOT iq_stValve.q_xOPN_DO, PT := tTimeOutDuration);


// Alarm reset
//////////////////////////////////////
ACT_ResetAlarms();

(*IO Mapping*)
ACT_IO();

// Log States and triggers
ACT_Logger();



(*FAST FAULT*)
FFO(i_xOK := xMPS_OK,
    i_xReset := i_xReset,
	i_xAutoReset :=TRUE,
    io_fbFFHWO := io_fbFFHWO);

ACTION ACT_IO:
(*inputs*)
iq_stValve.i_xOpnLS := 	i_xOpnLS;
iq_stValve.i_xClsLS:=	i_xClsLS;
iq_stValve.xEXT_OK := i_xEXT_OK;
iq_stValve.xOverrideMode := i_xOverrideMode;
(*outputs*)
q_xOPN_DO:= iq_stValve.q_xOPN_DO;

(*ILK Devices*)
iq_stValve.sIlkUSDeviceName := This^.i_stUSG.sPath;
iq_stValve.sIlkDSDeviceName := This^.i_stDSG.sPath;
END_ACTION

ACTION ACT_Logger:
// ILK logger

IF NOT (iq_stValve.xOPN_OK) AND (ePrevState = OPEN) AND NOT (TonOvrd.Q) THEN
 		fbLogger(sMsg:='Lost interlock ok bit while valve was open.', eSevr:=TcEventSeverity.Critical);  	
END_IF


//Positiong STATE Logger  
IF ePrevState <> iq_stValve.eState THEN
	  CASE iq_stValve.eState OF
		INVALID:
			fbLogger(sMsg:='Valve invalid position.', eSevr:=TcEventSeverity.Critical);
  		MOVING:
			fbLogger(sMsg:='Valve moving', eSevr:=TcEventSeverity.Warning);
		OPEN:
			fbLogger(sMsg:='Valve Open.', eSevr:=TcEventSeverity.Info);
		OPEN_F:
			fbLogger(sMsg:='Valve Open.', eSevr:=TcEventSeverity.Info);
		CLOSED:
			fbLogger(sMsg:='Valve closed.', eSevr:=TcEventSeverity.Info);
	  END_CASE
	  ePrevState := iq_stValve.eState;  
  END_IF
 
 //Pressure STATE Logger  
IF eVGCPrevState <> iq_stValve.eVGC_State THEN
	  CASE iq_stValve.eVGC_State OF
		Vented:
			 fbLogger(sMsg:='Vented', eSevr:=TcEventSeverity.Info);
  		AtVacuum:
			 fbLogger(sMsg:='Vacuum setpoint satisfied', eSevr:=TcEventSeverity.Info);
		ERR_DiffPress:
			 fbLogger(sMsg:='Potential accidental vent.', eSevr:=TcEventSeverity.Critical);
		ERR_LostVac:
			fbLogger(sMsg:='Unexpected loss of vacuum while valve was open or moving.', eSevr:=TcEventSeverity.Critical);
		ERR_ExtFault:
			 fbLogger(sMsg:='Lost external interlock while valve was open.', eSevr:=TcEventSeverity.Critical);
	  END_CASE
	  eVGCPrevState := iq_stValve.eVGC_State;  
  END_IF
  


// Log valve timeouts
tErrorPresent(CLK:=iq_stValve.bErrorPresent);
IF tErrorPresent.Q THEN fbLogger(sMsg:=iq_stValve.sErrorMessage, eSevr:=TcEventSeverity.Warning); END_IF

// Log valve open
tAction(CLK:= iq_stValve.q_xOPN_DO);
IF tAction.Q THEN fbLogger(sMsg:='Valve commanded open', eSevr:=TcEventSeverity.Info); END_IF

// Log override mode enabled
tOverrideActivated(CLK:= (tonOvrd.Q AND i_xOverrideMode));
IF tOverrideActivated.Q THEN fbLogger(sMsg:='Valve override mode activated', eSevr:=TcEventSeverity.Warning); END_IF
END_ACTION

ACTION ACT_PMPS:
bMoving := (iq_stValve.pv_xOPN_SW AND iq_stValve.i_xClsLS) XOR (NOT iq_stValve.pv_xOPN_SW AND i_xOpnLS);
bDone := (iq_stValve.pv_xOPN_SW AND iq_stValve.i_xOpnLS) XOR (NOT iq_stValve.pv_xOPN_SW AND i_xClsLS);
If (i_xIsAperture ) OR (iq_stValve.pv_xOPN_SW )THEN
	bptm.i_stRequestedAssertion := PMPS_GVL.cstFullBeam;
ELSE  bptm.i_stRequestedAssertion := PMPS_GVL.cstSafeBeam;
END_IF

bptm(fbArbiter:=fbArbiter,
     i_TransitionAssertionID:=i_nTransitionRootID+2,
     i_stTransitionAssertion:=PMPS_GVL.cstSafeBeam,
     i_nRequestedAssertionID:=i_nTransitionRootID+ BOOL_TO_UDINT( iq_stValve.pv_xOPN_SW),
     i_stRequestedAssertion:=,
     i_xMoving:=,//bMoving,
     i_xDoneMoving:= bDone,
     stCurrentBeamParameters:=PMPS_GVL.stCurrentBeamParameters,
     q_xTransitionAuthorized=>);
// Timeout
tBPTMtimeout(IN:= bMoving AND NOT bptm.q_xTransitionAuthorized, PT:=T#2S);
//xPMPS_OK := bptm.q_xTransitionAuthorized OR tBPTMtimeout.Q;
//xPMPS_OK := i_xPMPS_OK OR (bptm.q_xTransitionAuthorized OR tBPTMtimeout.Q); // Moved to FB, move it back after testing

//Timeout and clear request
IF (tBPTMtimeout.Q) THEN
	fbArbiter.RemoveRequest(bptm.i_TransitionAssertionID);
	fbArbiter.RemoveRequest(bptm.i_nRequestedAssertionID);
END_IF
END_ACTION

ACTION ACT_ResetAlarms:
iq_stValve.xERR_DifPres R= iq_stValve.pv_xAlmRst;
iq_stValve.xERR_SP R= iq_stValve.pv_xAlmRst;
iq_stValve.bErrorPresent R= iq_stValve.pv_xAlmRst;
iq_stValve.xERR_ExtFault R= iq_stValve.pv_xAlmRst;

IF ( iq_stValve.pv_xAlmRst) THEN
	iq_stValve.sErrorMessage :='';
	 iq_stValve.pv_xAlmRst := FALSE;
END_IF
END_ACTION

METHOD PUBLIC M_IsClosed : BOOL
VAR_INPUT
END_VAR
M_IsClosed := (This^.iq_stValve.eState = E_ValvePositionState.CLOSED);
END_METHOD

METHOD PUBLIC M_IsOpen : BOOL
VAR_INPUT
END_VAR
M_IsOpen := (This^.iq_stValve.eState = E_ValvePositionState.OPEN);
END_METHOD

// Use this Methode to Open or close the valve by setting the OPN_SW to the input value.
METHOD PUBLIC M_Set_OPN_SW : BOOL
VAR_INPUT
		value:BOOL;
END_VAR
This^.iq_stValve.pv_xOPN_SW := value;
END_METHOD

END_FUNCTION_BLOCK

// ---- POUs/MAIN.TcPOU
PROGRAM MAIN
VAR
	
	//Example implementation of an arbiter
    g_fbArbiter1    :   FB_Arbiter(1);
	 //g_fbArbiter2    :   FB_Arbiter(2);
	 // g_fbArbiter3    :   FB_Arbiter(3);
	//fbArbiterIO : FB_SubSysToArbiter_IO;
	  fbArbiterIO : FB_DummyArbIO;
 bTransC:BOOL;
  bTrans:BOOL;
 bClose:BOOL;
 bOpen:BOOL;
 bRemove:bool;

  bTrans2:BOOL;
 bClose2:BOOL;
 bOpen2:BOOL;
 ID:DWORD;
 
 //////////////////
 VFS_Interface:FB_VFS_Interface;
 VFS: FB_VFS;
  VFS2: FB_VFS;
 VGC_2S: FB_VGC_2S;
	xFirstPass: BOOL := TRUE;
	// For Persistent Data
	fbWritePersistentData           : WritePersistentData;
	rTempUpperLimit	:	REAL:=0;
	
	 PROFILER1     :PROFILER;
    ProfilerData  :PROFILERSTRUCT;
    a             :LREAL;
END_VAR

VAR PERSISTENT
    bSaved: BOOL;
    rUpperLimit	:	REAL;
END_VAR

(*On first PLC pass, load the persistent value into the structrue variable*)
IF (xFirstPass) THEN
	xFirstPass	:= FALSE;
	rTempUpperLimit := rUpperLimit;
END_IF
(*Check if a new value has been written in the structure variable copy it to the persistent variable*)
IF NOT (rTempUpperLimit= rUpperLimit) THEN
	rUpperLimit := rTempUpperLimit;
	//fbWritePersistentData(NETID:='', PORT:=851, START:=TRUE, TMOUT:=T#1s );
ELSE
     //fbWritePersistentData( START:=FALSE);
END_IF;

//rTempUpperLimit:=rTempUpperLimit+1;

PROFILER1(START := fbWritePersistentData.BUSY);



//FFO
g_FastFaultOutput1.Execute(bAutoReset:=TRUE);

//testing fast shutter
//VFS(i_xPMPS_OK:=TRUE , i_xExt_OK:=TRUE , i_sDevName:='vfs' , io_fbFFHWO:= g_FastFaultOutput1);
VFS_Interface(IG:= FEE_KMONO_GCC_01.IG , Veto_Valve:= VGC_2S.iq_stValve , iq_stValve=> , i_xVAC_FAULT_OK=> );
VFS(
	i_xPMPS_OK:= TRUE, 
	i_xExt_OK:= TRUE, 
	i_sDevName:= 'vfs', 
	i_xVeto_Enable:= TRUE, 
	io_fbFFHWO:= g_FastFaultOutput1 );
VGC_2S(
	i_stUSG:=  FEE_KMONO_GCC_01.IG, 
	i_stDSG:=  FEE_KMONO_GCC_01.IG, 
	i_xDis_DPIlk:= FALSE, 
	i_xPMPS_OK:= TRUE, 
	i_xEPS_OK:= TRUE, 
	i_xExt_OK:= TRUE, 
	i_xOverrideMode:= , 
	i_xReset:= , 
	i_xIsAperture:= FALSE, 
	i_sDevName:= 'DEV', 
	i_nTransitionRootID:=13 , 
	iq_stValve=> , 
	xMPS_OK=> , 
	io_fbFFHWO:= g_FastFaultOutput1, 
	fbArbiter:= g_fbArbiter1);




//testing pmps
g_FastFaultOutput2.Execute(bAutoReset:=TRUE);

//
//bTransC:= g_fbArbiter1.CheckRequestInPool(1010);//TransitionID
bTrans:= g_fbArbiter1.CheckRequestInPool(ID+2);//TransitionID
bClose:= g_fbArbiter1.CheckRequestInPool(ID);//Assertion Closed ID
bOpen:= g_fbArbiter1.CheckRequestInPool(ID+1);//Assertion Open ID
(*
bTrans2:= g_fbArbiter2.CheckRequestInPool(ID+2);//TransitionID
bClose2:= g_fbArbiter2.CheckRequestInPool(ID);//Assertion Closed ID
bOpen2:= g_fbArbiter2.CheckRequestInPool(ID+1);//Assertion Open ID*)
if (bRemove) THEN
	g_fbArbiter1.RemoveRequest(ID);
END_IF

//PMPS_GVL.stCurrentBeamParameters:= PMPS_GVL.cstFullBeam;// g_fbArbiter1.q_stBeamParams;
fbArbiterIO.AutoUpdateBP:=TRUE;
fbArbiterIO(LA := g_fbArbiter1, FFO := g_FastFaultOutput1, q_stSimulatedBPReadback => PMPS_GVL.stCurrentBeamParameters);
//g_fbArbiter1.ElevateRequest(g_fbArbiter2);
//valves
FEE_VGC_02(
	i_stUSG:= FEE_KMONO_GCC_01.IG, 
	i_stDSG:= FEE_KMONO_GCC_01.IG , 
	i_xDis_DPIlk:= FALSE,
	i_xEPS_OK :=TRUE,
	//i_xEPS_OPN_OK:= , 
	//i_xEPS_CLS_OK:= ,
	i_xPMPS_OK:= , 
	i_xExt_OK:= TRUE, 
	i_xOverrideMode:= , 
	i_xReset:= ,
	iq_stValve=>,
	xMPS_OK=> , 
	io_fbFFHWO:= g_FastFaultOutput1,
fbArbiter:= g_fbArbiter1,
i_nTransitionRootID:=7000 );

PMPS_VGC_01(
	i_stUSG:= FEE_KMONO_GCC_01.IG, 
	i_stDSG:= FEE_KMONO_GCC_01.IG , 
	i_xDis_DPIlk:= FALSE,
	i_xEPS_OK :=TRUE,
	//i_xEPS_OPN_OK:= , 
	//i_xEPS_CLS_OK:= ,
	i_xPMPS_OK:= , 
	i_xExt_OK:= TRUE, 
	i_xOverrideMode:= , 
	i_xReset:= ,
	iq_stValve=>,
	xMPS_OK=> , 
	io_fbFFHWO:= g_FastFaultOutput1,
fbArbiter:= g_fbArbiter1,
i_nTransitionRootID:=1000 );
PMPS_VGC_02(
	i_stUSG:= FEE_KMONO_GCC_01.IG, 
	i_stDSG:= FEE_KMONO_GCC_01.IG , 
	i_xDis_DPIlk:= FALSE,
	i_xEPS_OK :=TRUE,
	//i_xEPS_OPN_OK:= , 
	//i_xEPS_CLS_OK:= ,
	i_xPMPS_OK:= , 
	i_xExt_OK:= TRUE, 
	i_xOverrideMode:= , 
	i_xReset:= ,
	iq_stValve=>,
	xMPS_OK=> , 
	io_fbFFHWO:= g_FastFaultOutput1,
fbArbiter:= g_fbArbiter1,
i_nTransitionRootID:=2000 );

PMPS_VGC_03(
	i_stUSG:= FEE_KMONO_GCC_01.IG, 
	i_stDSG:= FEE_KMONO_GCC_01.IG , 
	i_xDis_DPIlk:= FALSE,
	i_xEPS_OK :=TRUE,
	//i_xEPS_OPN_OK:= , 
	//i_xEPS_CLS_OK:= ,
	i_xPMPS_OK:= , 
	i_xExt_OK:= TRUE, 
	i_xOverrideMode:= , 
	i_xReset:= ,
	iq_stValve=>,
	xMPS_OK=> , 
	io_fbFFHWO:= g_FastFaultOutput1,
fbArbiter:= g_fbArbiter1,
i_nTransitionRootID:=3000 );

PMPS_VGC_04(
	i_stUSG:= FEE_KMONO_GCC_01.IG, 
	i_stDSG:= FEE_KMONO_GCC_01.IG , 
	i_xDis_DPIlk:= FALSE,
	i_xEPS_OK :=TRUE,
	//i_xEPS_OPN_OK:= , 
	//i_xEPS_CLS_OK:= ,
	i_xPMPS_OK:= , 
	i_xExt_OK:= TRUE, 
	i_xOverrideMode:= , 
	i_xReset:= ,
	iq_stValve=>,
	xMPS_OK=> , 
	io_fbFFHWO:= g_FastFaultOutput1,
fbArbiter:= g_fbArbiter1,
i_nTransitionRootID:=4000 );

PMPS_VGC_05(
	i_stUSG:= FEE_KMONO_GCC_01.IG, 
	i_stDSG:= FEE_KMONO_GCC_01.IG , 
	i_xDis_DPIlk:= FALSE,
	i_xEPS_OK :=TRUE,
	//i_xEPS_OPN_OK:= , 
	//i_xEPS_CLS_OK:= ,
	i_xPMPS_OK:= , 
	i_xExt_OK:= TRUE, 
	i_xOverrideMode:= , 
	i_xReset:= ,
	iq_stValve=>,
	xMPS_OK=> , 
	io_fbFFHWO:= g_FastFaultOutput1,
fbArbiter:= g_fbArbiter1,
i_nTransitionRootID:=5000 );

PMPS_VGC_06(
	i_stUSG:= FEE_KMONO_GCC_01.IG, 
	i_stDSG:= FEE_KMONO_GCC_01.IG , 
	i_xDis_DPIlk:= FALSE,
	i_xEPS_OK :=TRUE,
	//i_xEPS_OPN_OK:= , 
	//i_xEPS_CLS_OK:= ,
	i_xPMPS_OK:= , 
	i_xExt_OK:= TRUE, 
	i_xOverrideMode:= , 
	i_xReset:= ,
	iq_stValve=>,
	xMPS_OK=> , 
	io_fbFFHWO:= g_FastFaultOutput1,
fbArbiter:= g_fbArbiter1,
i_nTransitionRootID:=6000 );

PMPS_VGC_08(
	i_stUSG:= FEE_KMONO_GCC_01.IG, 
	i_stDSG:= FEE_KMONO_GCC_01.IG , 
	i_xDis_DPIlk:= FALSE,
	i_xEPS_OK :=TRUE,
	//i_xEPS_OPN_OK:= , 
	//i_xEPS_CLS_OK:= ,
	i_xPMPS_OK:= , 
	i_xExt_OK:= TRUE, 
	i_xOverrideMode:= , 
	i_xReset:= ,
	iq_stValve=>,
	xMPS_OK=> , 
	io_fbFFHWO:= g_FastFaultOutput1,
fbArbiter:= g_fbArbiter1,
i_nTransitionRootID:=8000 );

PMPS_VGC_09(
	i_stUSG:= FEE_KMONO_GCC_01.IG, 
	i_stDSG:= FEE_KMONO_GCC_01.IG , 
	i_xDis_DPIlk:= FALSE,
	i_xEPS_OK :=TRUE,
	//i_xEPS_OPN_OK:= , 
	//i_xEPS_CLS_OK:= ,
	i_xPMPS_OK:= , 
	i_xExt_OK:= TRUE, 
	i_xOverrideMode:= , 
	i_xReset:= ,
	iq_stValve=>,
	xMPS_OK=> , 
	io_fbFFHWO:= g_FastFaultOutput1,
fbArbiter:= g_fbArbiter1,
i_nTransitionRootID:=9000 );

PMPS_VGC_10(
	i_stUSG:= FEE_KMONO_GCC_01.IG, 
	i_stDSG:= FEE_KMONO_GCC_01.IG , 
	i_xDis_DPIlk:= FALSE,
	i_xEPS_OK :=TRUE,
	//i_xEPS_OPN_OK:= , 
	//i_xEPS_CLS_OK:= ,
	i_xPMPS_OK:= , 
	i_xExt_OK:= TRUE, 
	i_xOverrideMode:= , 
	i_xReset:= ,
	iq_stValve=>,
	xMPS_OK=> , 
	io_fbFFHWO:= g_FastFaultOutput1,
fbArbiter:= g_fbArbiter1,
i_nTransitionRootID:=10000 );
(*
PMPS_VGC_11(
	i_stUSG:= FEE_KMONO_GCC_01.IG, 
	i_stDSG:= FEE_KMONO_GCC_01.IG , 
	i_xDis_DPIlk:= FALSE,
	i_xEPS_OK :=TRUE,
	//i_xEPS_OPN_OK:= , 
	//i_xEPS_CLS_OK:= ,
	i_xPMPS_OK:= , 
	i_xExt_OK:= TRUE, 
	i_xOverrideMode:= , 
	i_xReset:= ,
	iq_stValve=>,
	xMPS_OK=> , 
	io_fbFFHWO:= g_FastFaultOutput1,
fbArbiter:= g_fbArbiter2,
i_nTransitionRootID:=11000 );*)



// gauges interlocking VGC_02 using the same gauge for the purpose of this test
FEE_KMONO_GPI_01(PG=>);
FEE_KMONO_GCC_01(PG:=FEE_KMONO_GPI_01.PG);

// Following are function block for the rest of the beamline devices
FEE_KMONO_PIP_01(i_stGauge:= FEE_KMONO_GPI_01.PG);
FEE_GPI_03(PG=>);
FEE_GCC_03(PG:=FEE_KMONO_GPI_01.PG);

FEE_PIP_02(i_stGauge:= FEE_GCC_03.IG);

FEE_M1L_GPI_01(PG=>);
FEE_M1L_GCC_01(PG:=FEE_M1L_GPI_01.PG);
FEE_M1L_PIP_01(i_stGauge:= FEE_M1L_GCC_01.IG);

FEE_GPI_04(PG=>);
FEE_GCC_04(PG:=FEE_GPI_04.PG);
FEE_PIP_03(i_stGauge:= FEE_GCC_04.IG);

//PTM
PTM_Agilent(I_xExtIlkOk := TRUE, i_stGauge:= FEE_GPI_04.PG, i_rMaxBackingPressure := 2);

END_PROGRAM
